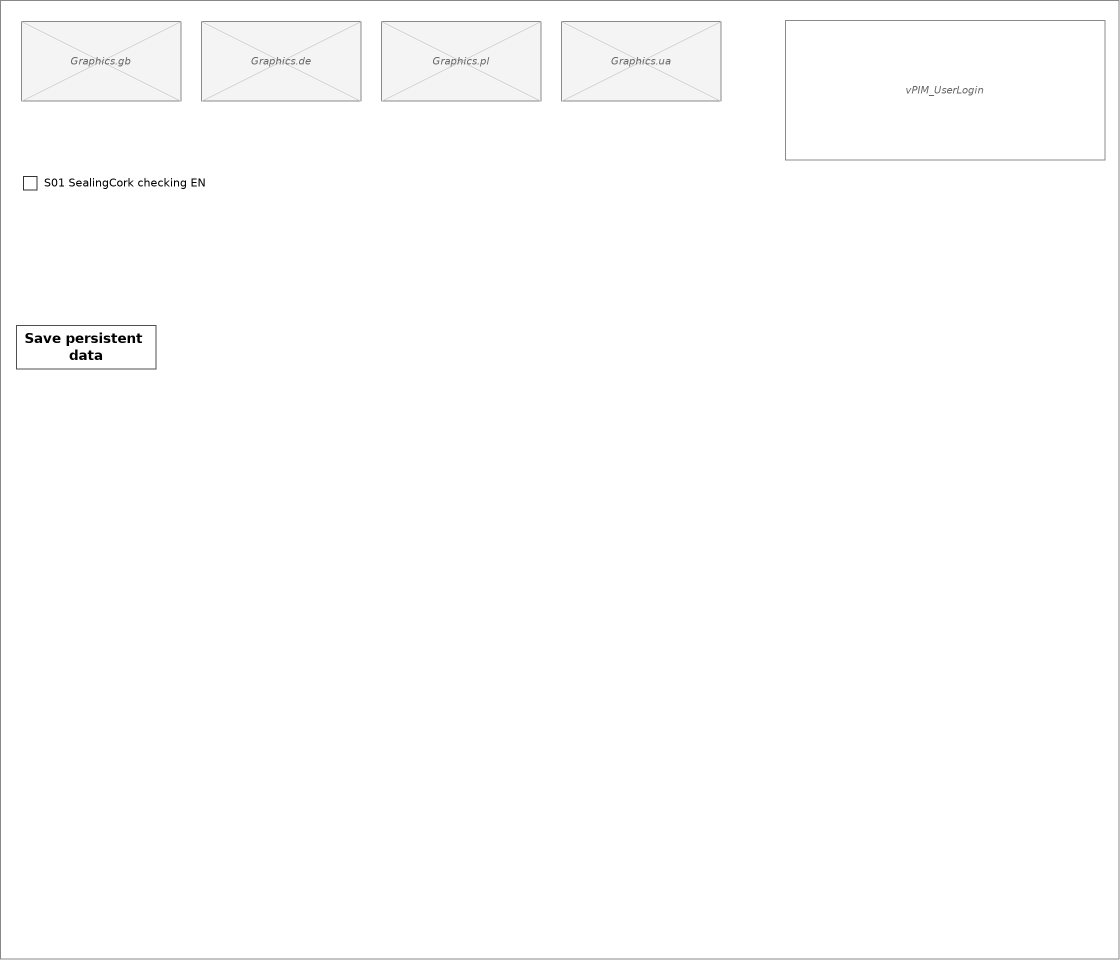
VISUALIZATION vGlobalSettings  // 1120x960
    Image (21,21 160x80), image: Graphics.gb
        OnMouseClick: ChangeLanguage ChangeLanguage=en
    Image (201,21 160x80), image: Graphics.de
        OnMouseClick: ChangeLanguage ChangeLanguage=de
    Image (381,21 160x80), image: Graphics.pl
        OnMouseClick: ChangeLanguage ChangeLanguage=pl
    Image (561,21 160x80), image: Graphics.ua
        OnMouseClick: ChangeLanguage ChangeLanguage=ua
    Frame (785,20 320x140)
        shows vPIM_UserLogin(fbPIM := GVL.fbUserLogin)
    Rectangle (16,325 140x44), "Save persistent data"
        tap GVL_Aircom.bWritePersistent
    Checkbox (21,168 291x30), "S01 SealingCork checking EN", variable: MAIN.fbS01_KeyencePNVisSens.bEnCheck
END_VISUALIZATION

(* stored: Version 1.1.0.1, ProductVersion 3.1.4024.13
   Visu vGlobalSettings: Id {9665561a-d695-49f7-986e-9717bd7e751c} *)
